// TIA Portal V18 export
TYPE "Starter_HPU_IO_In"
   STRUCT
      Slot2 { ExternalWritable := 'False'} : "TM_Count_Man_In";
      Slot3 { ExternalWritable := 'False'} : "DI16x24V_In";
      Slot4 { ExternalWritable := 'False'} : "DI16x24V_In";
      Slot5 { S7_SetPoint := 'True'} : "AI8xU_In";
      Slot6 { ExternalWritable := 'False'} : "AI8xI_In";
      Slot7 { ExternalWritable := 'False'} : "TM_Pulse_2x24_In";
      Slot8 { S7_SetPoint := 'True'} : "TM_Pulse_2x24_In";
      Slot9 { S7_SetPoint := 'True'} : "TM_Pulse_2x24_In";
   END_STRUCT;
END_TYPE
